// TIA Portal V17 export
// export: Created 2023-04-04T13:27:30.4188586Z, ExportSetting WithDefaults, DisplayName Totally Integrated Automation Portal, DisplayVersion V17, DisplayName TIA Portal Openness, DisplayVersion V17, DisplayName TIA Portal Version Control Interface, DisplayVersion V17, DisplayName STEP 7 Professional, DisplayVersion V17, DisplayName STEP 7 Safety, DisplayVersion V17, DisplayName WinCC Advanced, DisplayVersion V17
VAR_GLOBAL   // PLC tag table "SSC - Sensor-Station Camera"
   IX_SSC_RefSwitchVerticalAxis_I1 AT %I4.0 : Bool;   // SSC - I1 = Reference switch vertical axis   {ExternalAccessible false, ExternalVisible false, ExternalWritable false}
   IX_SSC_RefSwitchHorizontalAxis_I2 AT %I4.1 : Bool;   // SSC - I2 = Reference switch horizontal axis   {ExternalAccessible false, ExternalVisible false, ExternalWritable false}
   IX_SSC_LightBarrierStorage_I3 AT %I4.3 : Bool;   // SSC - I3 = Light barrier inlet   {ExternalAccessible false, ExternalVisible false, ExternalWritable false}
   IX_SSC_LightBarrierOutsourcing_I4 AT %I4.2 : Bool;   // SSC - I4 = Light barrier behind color sensor   {ExternalAccessible false, ExternalVisible false, ExternalWritable false}
   IW_SSC_ColorSensor_A1 AT %IW9 : Word;   // SSC - A1 = Color sensor   {ExternalAccessible false, ExternalVisible false, ExternalWritable false}
   IX_SSC_EncoderVerticalAxisImp1_B1 AT %I5.3 : Bool;   // SSC - B1 = Encoder vertical axis imulse 1   {ExternalAccessible false, ExternalVisible false, ExternalWritable false}
   IX_SSC_EncoderVerticalAxisImp2_B2 AT %I5.7 : Bool;   // SSC - B2 = Encoder vertical axis imulse 2   {ExternalAccessible false, ExternalVisible false, ExternalWritable false}
   IX_SSC_EncoderHorizontalAxisImp1_B3 AT %I6.3 : Bool;   // SSC - B3 = Encoder horizontal axis imulse 1   {ExternalAccessible false, ExternalVisible false, ExternalWritable false}
   IX_SSC_EncoderHorizontalAxisImp2_B4 AT %I6.7 : Bool;   // SSC - B4 = Encoder horizontal axis imulse 2   {ExternalAccessible false, ExternalVisible false, ExternalWritable false}
   QX_SSC_M1_VerticalAxisUp_Q1 AT %Q6.0 : Bool;   // SSC - Q1 = Motor M1 vertical axis up   {ExternalAccessible false, ExternalVisible false, ExternalWritable false}
   QX_SSC_M1_VerticalAxisDown_Q2 AT %Q6.1 : Bool;   // SSC - Q2 = Motor M1 vertical axis down   {ExternalAccessible false, ExternalVisible false, ExternalWritable false}
   QX_SSC_M2_HorizontalAxisClockwise_Q3 AT %Q6.3 : Bool;   // SSC - Q3 = Motor M2 horizontal axis backward   {ExternalAccessible false, ExternalVisible false, ExternalWritable false}
   QX_SSC_M2_HorizontalAxisCounterclockwise_Q4 AT %Q6.2 : Bool;   // SSC - Q4 = Motor M2 horizontal axis forward   {ExternalAccessible false, ExternalVisible false, ExternalWritable false}
   QX_SSC_LED_Green_Q5 AT %Q6.4 : Bool;   // SSC - Q5 = LED Green   {ExternalAccessible false, ExternalVisible false, ExternalWritable false}
   QX_SSC_LED_Yellow_Q6 AT %Q6.5 : Bool;   // SSC - Q6 = LED Yellow   {ExternalAccessible false, ExternalVisible false, ExternalWritable false}
   QX_SSC_LED_Red_Q7 AT %Q6.6 : Bool;   // SSC - Q7 = LED Red   {ExternalAccessible false, ExternalVisible false, ExternalWritable false}
   QX_SSC_LED_Red_Online_Q8 AT %Q6.7 : Bool;   // SSC - Q8 = LED Red Online   {ExternalAccessible false, ExternalVisible false, ExternalWritable false}
   QW_SSC_PWM_Vertical_M1 AT %QW27 : Int;   // SSC = PWM Motor M1 vertical axis   {ExternalAccessible false, ExternalVisible false, ExternalWritable false}
   QW_SSC_PWM_Horizontal_M2 AT %QW29 : Int;   // SSC = PWM Motor M2 horizontal axis   {ExternalAccessible false, ExternalVisible false, ExternalWritable false}
END_VAR
